// TIA Portal V18 export
// export: Created 2026-06-23T08:49:31.3755169Z, ExportSetting WithDefaults, DisplayName Totally Integrated Automation Portal, DisplayVersion V18, DisplayName TIA Portal Openness, DisplayVersion V18, DisplayName TIA Portal Version Control Interface, DisplayVersion V18, DisplayName STEP 7 Professional, DisplayVersion V18, DisplayName STEP 7 Safety, DisplayVersion V18, DisplayName WinCC Professional, DisplayVersion V18
FUNCTION "FC_HMI_Animation_PLC2" : Void   // FC61, LAD
{ S7_Optimized_Access := 'TRUE' }
VERSION : 0.1
// stored: AutoNumber true, IsIECCheckEnabled false, SetENOAutomatically false, UDAEnableTagReadback false
BEGIN

REGION Network 1: Cánh khuấy Bồn 3: Tăng khung hình khi chạy
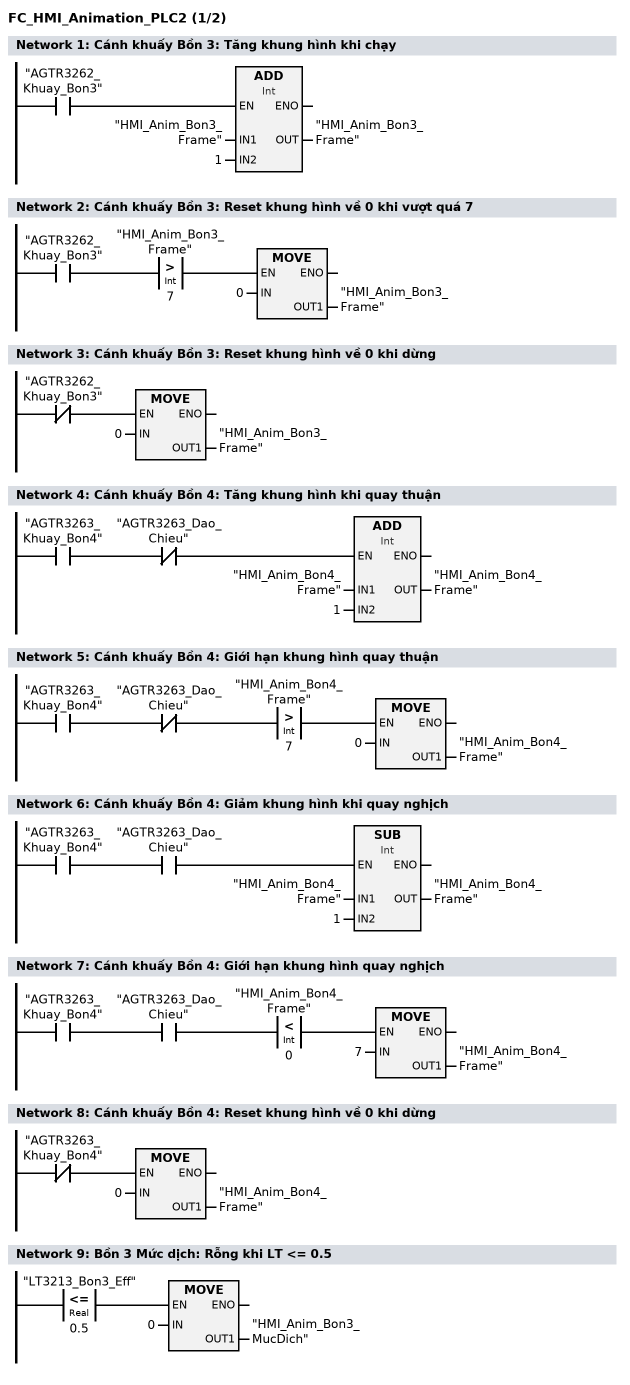
   RUNG wire#powerrail
      Contact( "AGTR3262_Khuay_Bon3" )
      { S7_Templates := "SrcType := Int"; S7_GenerateENO := "TRUE" } Add(in1 := "HMI_Anim_Bon3_Frame", in2 := 1, out => "HMI_Anim_Bon3_Frame")
   END_RUNG
   // the same network as SCL:
   IF "AGTR3262_Khuay_Bon3" THEN "HMI_Anim_Bon3_Frame" := "HMI_Anim_Bon3_Frame" + 1; END_IF;
END_REGION

REGION Network 2: Cánh khuấy Bồn 3: Reset khung hình về 0 khi vượt quá 7
   RUNG wire#powerrail
      Contact( "AGTR3262_Khuay_Bon3" )
      { S7_Templates := "SrcType := Int" } GT_Contact(in1 := "HMI_Anim_Bon3_Frame", in2 := 7)
      { S7_GenerateENO := "TRUE" } Move(in := 0, out1 => "HMI_Anim_Bon3_Frame")
   END_RUNG
   // the same network as SCL:
   IF "AGTR3262_Khuay_Bon3" AND ("HMI_Anim_Bon3_Frame" > 7) THEN "HMI_Anim_Bon3_Frame" := 0; END_IF;
END_REGION

REGION Network 3: Cánh khuấy Bồn 3: Reset khung hình về 0 khi dừng
   RUNG wire#powerrail
      I_Contact( "AGTR3262_Khuay_Bon3" )
      { S7_GenerateENO := "TRUE" } Move(in := 0, out1 => "HMI_Anim_Bon3_Frame")
   END_RUNG
   // the same network as SCL:
   IF NOT "AGTR3262_Khuay_Bon3" THEN "HMI_Anim_Bon3_Frame" := 0; END_IF;
END_REGION

REGION Network 4: Cánh khuấy Bồn 4: Tăng khung hình khi quay thuận
   RUNG wire#powerrail
      Contact( "AGTR3263_Khuay_Bon4" )
      I_Contact( "AGTR3263_Dao_Chieu" )
      { S7_Templates := "SrcType := Int"; S7_GenerateENO := "TRUE" } Add(in1 := "HMI_Anim_Bon4_Frame", in2 := 1, out => "HMI_Anim_Bon4_Frame")
   END_RUNG
   // the same network as SCL:
   IF "AGTR3263_Khuay_Bon4" AND NOT "AGTR3263_Dao_Chieu" THEN
       "HMI_Anim_Bon4_Frame" := "HMI_Anim_Bon4_Frame" + 1;
   END_IF;
END_REGION

REGION Network 5: Cánh khuấy Bồn 4: Giới hạn khung hình quay thuận
   RUNG wire#powerrail
      Contact( "AGTR3263_Khuay_Bon4" )
      I_Contact( "AGTR3263_Dao_Chieu" )
      { S7_Templates := "SrcType := Int" } GT_Contact(in1 := "HMI_Anim_Bon4_Frame", in2 := 7)
      { S7_GenerateENO := "TRUE" } Move(in := 0, out1 => "HMI_Anim_Bon4_Frame")
   END_RUNG
   // the same network as SCL:
   IF "AGTR3263_Khuay_Bon4" AND NOT "AGTR3263_Dao_Chieu" AND ("HMI_Anim_Bon4_Frame" > 7) THEN
       "HMI_Anim_Bon4_Frame" := 0;
   END_IF;
END_REGION

REGION Network 6: Cánh khuấy Bồn 4: Giảm khung hình khi quay nghịch
   RUNG wire#powerrail
      Contact( "AGTR3263_Khuay_Bon4" )
      Contact( "AGTR3263_Dao_Chieu" )
      { S7_Templates := "SrcType := Int"; S7_GenerateENO := "TRUE" } Sub(in1 := "HMI_Anim_Bon4_Frame", in2 := 1, out => "HMI_Anim_Bon4_Frame")
   END_RUNG
   // the same network as SCL:
   IF "AGTR3263_Khuay_Bon4" AND "AGTR3263_Dao_Chieu" THEN
       "HMI_Anim_Bon4_Frame" := "HMI_Anim_Bon4_Frame" - 1;
   END_IF;
END_REGION

REGION Network 7: Cánh khuấy Bồn 4: Giới hạn khung hình quay nghịch
   RUNG wire#powerrail
      Contact( "AGTR3263_Khuay_Bon4" )
      Contact( "AGTR3263_Dao_Chieu" )
      { S7_Templates := "SrcType := Int" } LT_Contact(in1 := "HMI_Anim_Bon4_Frame", in2 := 0)
      { S7_GenerateENO := "TRUE" } Move(in := 7, out1 => "HMI_Anim_Bon4_Frame")
   END_RUNG
   // the same network as SCL:
   IF "AGTR3263_Khuay_Bon4" AND "AGTR3263_Dao_Chieu" AND ("HMI_Anim_Bon4_Frame" < 0) THEN
       "HMI_Anim_Bon4_Frame" := 7;
   END_IF;
END_REGION

REGION Network 8: Cánh khuấy Bồn 4: Reset khung hình về 0 khi dừng
   RUNG wire#powerrail
      I_Contact( "AGTR3263_Khuay_Bon4" )
      { S7_GenerateENO := "TRUE" } Move(in := 0, out1 => "HMI_Anim_Bon4_Frame")
   END_RUNG
   // the same network as SCL:
   IF NOT "AGTR3263_Khuay_Bon4" THEN "HMI_Anim_Bon4_Frame" := 0; END_IF;
END_REGION

REGION Network 9: Bồn 3 Mức dịch: Rỗng khi LT <= 0.5
   RUNG wire#powerrail
      { S7_Templates := "SrcType := Real" } LE_Contact(in1 := "LT3213_Bon3_Eff", in2 := 0.5)
      { S7_GenerateENO := "TRUE" } Move(in := 0, out1 => "HMI_Anim_Bon3_MucDich")
   END_RUNG
   // the same network as SCL:
   IF "LT3213_Bon3_Eff" <= 0.5 THEN "HMI_Anim_Bon3_MucDich" := 0; END_IF;
END_REGION

REGION Network 10: Bồn 3 Mức dịch: Mức 40% khi 0.5 < LT < 50.0
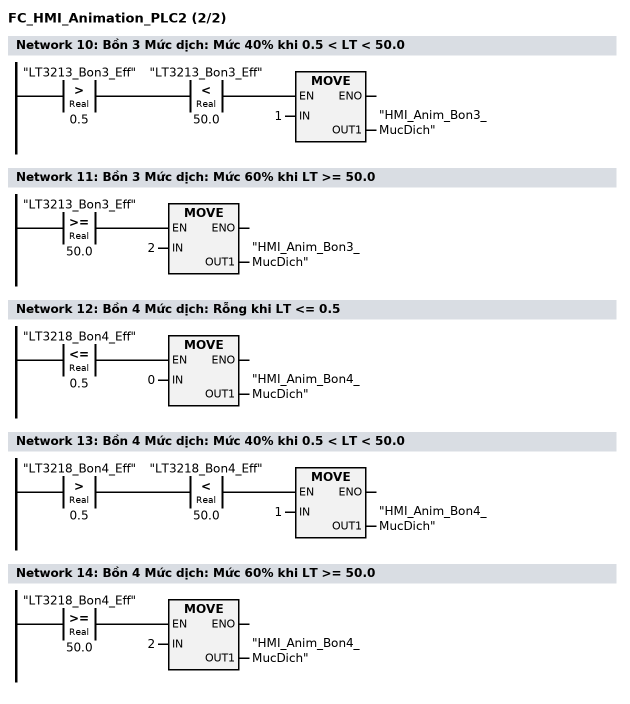
   RUNG wire#powerrail
      { S7_Templates := "SrcType := Real" } GT_Contact(in1 := "LT3213_Bon3_Eff", in2 := 0.5)
      { S7_Templates := "SrcType := Real" } LT_Contact(in1 := "LT3213_Bon3_Eff", in2 := 50.0)
      { S7_GenerateENO := "TRUE" } Move(in := 1, out1 => "HMI_Anim_Bon3_MucDich")
   END_RUNG
   // the same network as SCL:
   IF ("LT3213_Bon3_Eff" > 0.5) AND ("LT3213_Bon3_Eff" < 50.0) THEN "HMI_Anim_Bon3_MucDich" := 1; END_IF;
END_REGION

REGION Network 11: Bồn 3 Mức dịch: Mức 60% khi LT >= 50.0
   RUNG wire#powerrail
      { S7_Templates := "SrcType := Real" } GE_Contact(in1 := "LT3213_Bon3_Eff", in2 := 50.0)
      { S7_GenerateENO := "TRUE" } Move(in := 2, out1 => "HMI_Anim_Bon3_MucDich")
   END_RUNG
   // the same network as SCL:
   IF "LT3213_Bon3_Eff" >= 50.0 THEN "HMI_Anim_Bon3_MucDich" := 2; END_IF;
END_REGION

REGION Network 12: Bồn 4 Mức dịch: Rỗng khi LT <= 0.5
   RUNG wire#powerrail
      { S7_Templates := "SrcType := Real" } LE_Contact(in1 := "LT3218_Bon4_Eff", in2 := 0.5)
      { S7_GenerateENO := "TRUE" } Move(in := 0, out1 => "HMI_Anim_Bon4_MucDich")
   END_RUNG
   // the same network as SCL:
   IF "LT3218_Bon4_Eff" <= 0.5 THEN "HMI_Anim_Bon4_MucDich" := 0; END_IF;
END_REGION

REGION Network 13: Bồn 4 Mức dịch: Mức 40% khi 0.5 < LT < 50.0
   RUNG wire#powerrail
      { S7_Templates := "SrcType := Real" } GT_Contact(in1 := "LT3218_Bon4_Eff", in2 := 0.5)
      { S7_Templates := "SrcType := Real" } LT_Contact(in1 := "LT3218_Bon4_Eff", in2 := 50.0)
      { S7_GenerateENO := "TRUE" } Move(in := 1, out1 => "HMI_Anim_Bon4_MucDich")
   END_RUNG
   // the same network as SCL:
   IF ("LT3218_Bon4_Eff" > 0.5) AND ("LT3218_Bon4_Eff" < 50.0) THEN "HMI_Anim_Bon4_MucDich" := 1; END_IF;
END_REGION

REGION Network 14: Bồn 4 Mức dịch: Mức 60% khi LT >= 50.0
   RUNG wire#powerrail
      { S7_Templates := "SrcType := Real" } GE_Contact(in1 := "LT3218_Bon4_Eff", in2 := 50.0)
      { S7_GenerateENO := "TRUE" } Move(in := 2, out1 => "HMI_Anim_Bon4_MucDich")
   END_RUNG
   // the same network as SCL:
   IF "LT3218_Bon4_Eff" >= 50.0 THEN "HMI_Anim_Bon4_MucDich" := 2; END_IF;
END_REGION
END_FUNCTION
